{attribute 'qualified_only'}
VAR_GLOBAL

END_VAR
VAR_GLOBAL CONSTANT
	maxInputEventListeners: INT := 64;
	maxInputEventsPerNotification: INT := 4;
END_VAR

(* stored: Version 1.1.0.1, ProductVersion 3.1.4024.11
   GVL GVL_DALIBridge: Id {47208f56-9ae3-4f64-a4ef-661236969cfc} *)
